ADAPTER L3_ASetup
  (* Standard: 61499-1 *)
  (* Version 0.0, 2008-04-22, EQUEROL, UJI *)
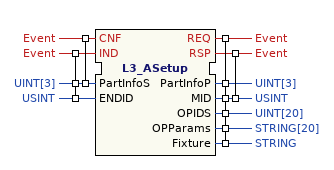
  EVENT_INPUT
    CNF WITH PartInfoS; (* Setup assignation confirmation *)
    IND WITH PartInfoS, ENDID; (* Completed setup indication *)
  END_EVENT
  EVENT_OUTPUT
    REQ WITH OPIDS, PartInfoP, MID, OPParams, Fixture; (* Plugin request to assign a setup *)
    RSP WITH MID; (* Completed setup indication treatement resposne *)
  END_EVENT
  VAR_INPUT
    PartInfoS : ARRAY [0..2] OF UINT; (* Part ID, Part Family, Part Type *)
    ENDID : USINT; (* Setup execution returned code *)
  END_VAR
  VAR_OUTPUT
    PartInfoP : ARRAY [0..2] OF UINT; (* PartID, Part Family, Part Type *)
    MID : USINT; (* Destination machine identifier *)
    OPIDS : ARRAY [0..19] OF UINT; (* Operations Identifiers *)
    OPParams : ARRAY [0..19] OF STRING; (* Operation parameters *)
    Fixture : STRING; (* Fixture to be used with the setup *)
  END_VAR
  SERVICE SOCKET/PLUG
    SEQUENCE request_confirm
      SOCKET.REQ(REQD) -> PLUG.REQ(REQD);
      PLUG.CNF(CNFD) -> SOCKET.CNF(CNFD);
    END_SEQUENCE
    SEQUENCE indication_response
      PLUG.IND(INDD) -> SOCKET.IND(INDD);
      SOCKET.RSP(RSPD) -> PLUG.RSP(RSPD);
    END_SEQUENCE
  END_SERVICE
END_ADAPTER
